Staubli VAL3: remErrFar.pgx

program remErrFar(string& sReturn[] (dimensions=1))
begin
  // Error raised when we try to move to a point that is too far
  //
  logMsg("call remErrFar")
  sReturn="ERROR 303: Move distance above limit."
  putln(sReturn)
  logMsg(sReturn)
end
